TYPE Torr : REAL; END_TYPE

(* stored: Version 1.1.0.1, ProductVersion 3.1.4024.4
   DUT Torr: Id {09d322ec-e4c8-44c9-9957-50369defddfd} *)
